TYPE ST_TimeStamp :
(**************************************************************************************
 * 	Application		:	BoxControl Framework
 *	Revision		:	$Revision: 404529 $
 *	Revision date	:	$Date: 2018-04-23 08:21:38 +0200 (Mo., 23 Apr 2018) $
 *	Last changed by	:	$Author: b7bolm $
 *	URL				:	$URL: http://almscdc.swisslog.com/repo/SWPD/Development/BoxControlFramework/20_Release/trunk/01_Software/BCF/BCF/JumpStart/20_Product/10_App/10_Base/10_Lib/10_Conv/01_DUTs/ST_TimeStamp.TcDUT $
 *
 *	Purpose			:	TU Data Time Stamp
 *
 * ------------------------------------------------------------------------------------
 *	Copyright Swisslog [IP AG], Switzerland. All rights reserved.
 * 
 * ------------------------------------------------------------------------------------
 *	
 * 	Revision History: 
 *
 * VERSION DATE         INITIALS     DESCRIPTION
 * 0.0     DD.MM.YYYY   (name)       (explain customized modifications)
 *
 **************************************************************************************)
STRUCT
	eInsertFunctionNumber		: E_FunctionNumber			:= 0;	// Inserted function number
	InsertZoneNumber			: INT						:= 0;	// Inserted zone number
	InsertDateTime				: Tc2_Utilities.TIMESTRUCT;			// Date and time of the insert 
END_STRUCT
END_TYPE

(* stored: Version 1.1.0.1, ProductVersion 3.1.4024.4
   DUT ST_TimeStamp: Id {1480c98a-0117-4c30-aaeb-5384b7e52be9} *)
